// Mitsubishi GX Works2 project: 0129 실린더 2개 단속   PLC: Q03UDV

PROGRAM MAIN
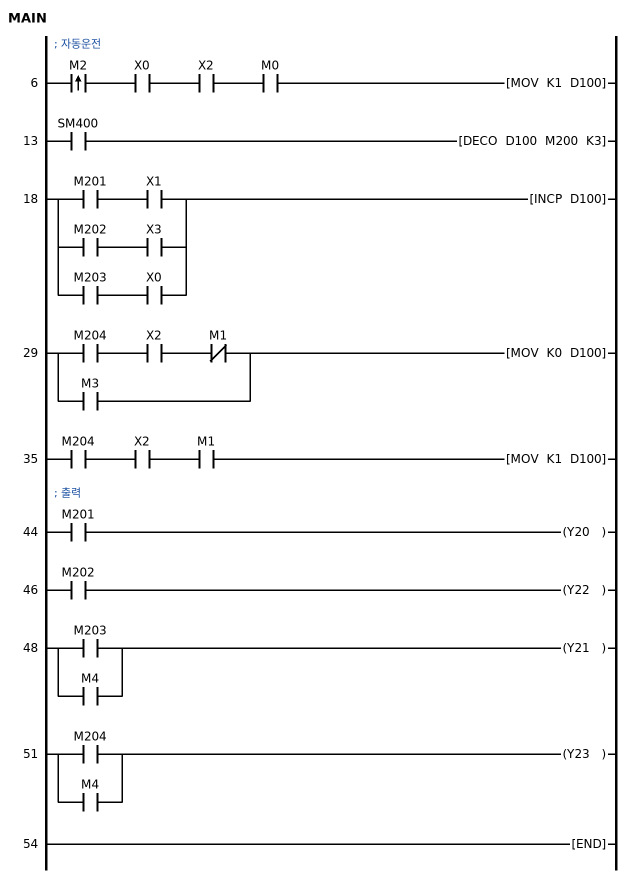
; 자동운전
6     LDP     M2
      AND     X0
      AND     X2
      AND     M0
      MOV     K1 D100
13    LD      SM400
      DECO    D100 M200 K3
18    LD      M201
      AND     X1
      LD      M202
      AND     X3
      ORB
      LD      M203
      AND     X0
      ORB
      INCP    D100
29    LD      M204
      AND     X2
      ANI     M1
      OR      M3
      MOV     K0 D100
35    LD      M204
      AND     X2
      AND     M1
      MOV     K1 D100
; 출력
44    LD      M201
      OUT     Y20
46    LD      M202
      OUT     Y22
48    LD      M203
      OR      M4
      OUT     Y21
51    LD      M204
      OR      M4
      OUT     Y23
54    END
END_PROGRAM
